FUNCTION_BLOCK E_RDELAY (* Reloadable delayed propagation of an event-Cancellable *)
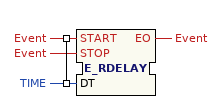
  EVENT_INPUT
    START WITH DT; (* Begin/Reset Delay *)
    STOP; (* Cancel Delay *)
  END_EVENT
  EVENT_OUTPUT
    EO; (* Delayed Event *)
  END_EVENT
  VAR_INPUT
    DT : TIME; (* Delay Time *)
  END_VAR
  SERVICE E_DELAY/RESOURCE (* Reloadable delayed propagation of an event-Cancellable *)
    SEQUENCE event_delay
      E_DELAY.START(DT) -> E_DELAY.EO();
    END_SEQUENCE
    SEQUENCE delay_canceled
      E_DELAY.START(DT);
      E_DELAY.STOP();
    END_SEQUENCE
    SEQUENCE no_multiple_delay
      E_DELAY.START(DT);
      E_DELAY.START(DT);
      -> E_DELAY.EO();
    END_SEQUENCE
  END_SERVICE
END_FUNCTION_BLOCK
